// SIMATIC STEP 7 (V5.x) project Actuadores_Lineales

SYMBOL_TABLE
"DERECHA"	I 8.1	BOOL	// Push Button direccion derecha
"IZQUIERDA"	I 8.2	BOOL	// Push Button direccion izquierda
"FIN"	I 8.3	BOOL	// Final de carrera
"INI"	I 8.4	BOOL	// Final de carrear inicio
"DIRm"	M 1.0	BOOL	// Direccion memoria
"STEPm"	M 1.1	BOOL
"DIR"	Q 12.0	BOOL
"STEP"	Q 12.1	BOOL
END_SYMBOL_TABLE
